(* Logix 5000 project; controller reto3 vendor 1 type 14 code 156 rev 30.11; software revision 30.00 *)

TASK MainTask (continuous, watchdog 500 ms) : MainProgram

MODULES
   Local : vendor 1 type 14 code 156 (Compact 0, rev 30.11)
      DI_4 : 1769-IQ16 (Compact 4, rev 1.1, Input RPI 20 ms)
      D0_5 : vendor 1 type 7 code 86 (Compact 5, rev 2.1, Output RPI 20 ms)
END_MODULES

ADD_ON_INSTRUCTION ACT_DE   (* revision 1.0 *)
VAR_INPUT
   PRENDER_DE : BOOL; {required}
END_VAR
VAR_IN_OUT
   CIERRE_DE : BOOL; {required}
   APERTURA_DE : BOOL; {required}
END_VAR
VAR
   TON_APERTURA_DE : TIMER := (PRE := 200); {access None}
   E_PRENDER : BOOL;
END_VAR

ROUTINE Logic   (* ladder *)
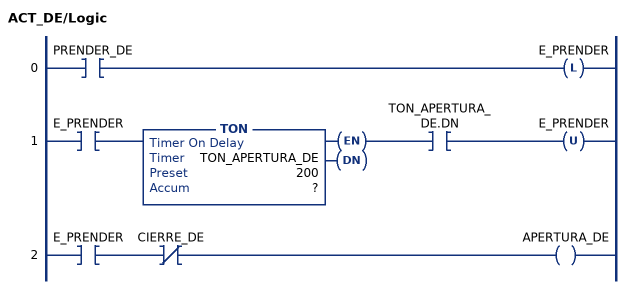
   0: XIC(PRENDER_DE)OTL(E_PRENDER);
   1: XIC(E_PRENDER)TON(TON_APERTURA_DE,?,?)XIC(TON_APERTURA_DE.DN)OTU(E_PRENDER);
   2: XIC(E_PRENDER)XIO(CIERRE_DE)OTE(APERTURA_DE);
END_ROUTINE
END_ADD_ON_INSTRUCTION

ADD_ON_INSTRUCTION CIE_DE   (* revision 1.0 *)
VAR_INPUT
   APAGAR_DE : BOOL; {required}
END_VAR
VAR_IN_OUT
   APERTURA_DE : BOOL; {required}
   CIERRE_DE : BOOL; {required}
END_VAR
VAR
   E_APAGAR : BOOL; {access None}
   TON_CIERRE_dE : TIMER := (PRE := 300); {access None}
END_VAR

ROUTINE Logic   (* ladder *)
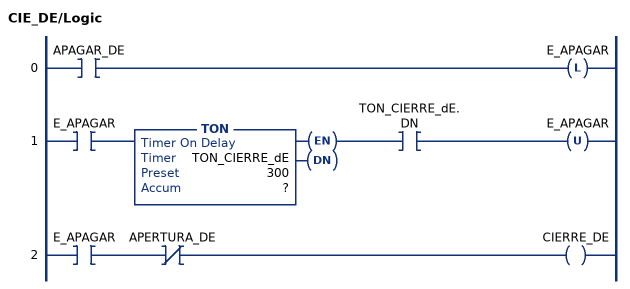
   0: XIC(APAGAR_DE)OTL(E_APAGAR);
   1: XIC(E_APAGAR)TON(TON_CIERRE_dE,?,?)XIC(TON_CIERRE_dE.DN)OTU(E_APAGAR);
   2: XIC(E_APAGAR)XIO(APERTURA_DE)OTE(CIERRE_DE);
END_ROUTINE
END_ADD_ON_INSTRUCTION

ADD_ON_INSTRUCTION COUNTERS   (* revision 1.0 *)
VAR_IN_OUT
   COUNTER_1 : DINT; {required}
END_VAR
VAR_INPUT
   OUT : BOOL; {required}
END_VAR
VAR_IN_OUT
   COUNTER_2 : DINT; {required}
   COUNTER_3 : DINT; {required}
END_VAR
VAR_INPUT
   IN_1 : BOOL; {access None, required}
   IN_2 : BOOL; {access None, required}
   IN_3 : BOOL; {access None, required}
END_VAR
VAR
   CUP_1 : BOOL; {access None}
   CUP_2 : BOOL; {access None}
   CUP_3 : BOOL; {access None}
   OSF_OB1 : BOOL; {access None}
   OSF_SB1 : BOOL; {access None}
   OSF_OB2 : BOOL; {access None}
   OSF_SB2 : BOOL; {access None}
   OSF_OB3 : BOOL; {access None}
   OSF_SB3 : BOOL; {access None}
   OP : BOOL; {access None}
END_VAR

ROUTINE Logic   (* ladder *)
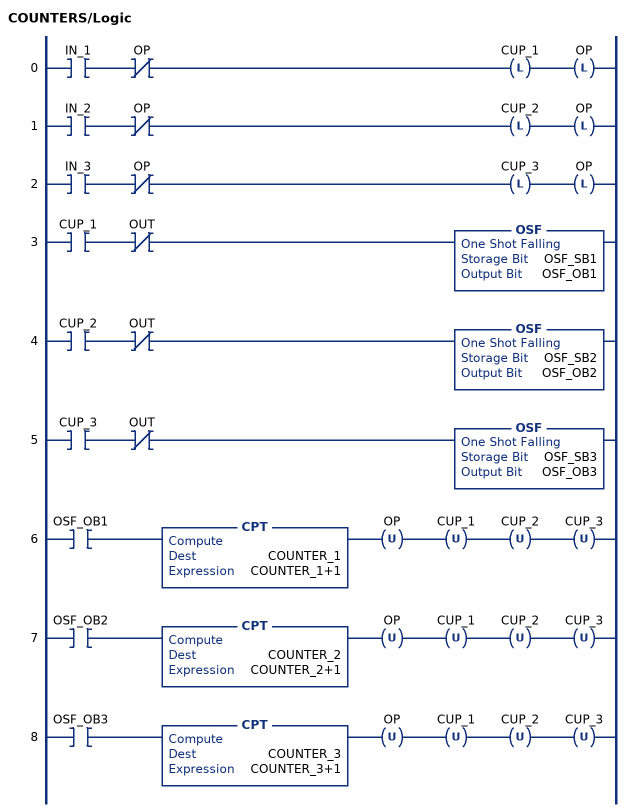
   0: XIC(IN_1)XIO(OP)OTL(CUP_1)OTL(OP);
   1: XIC(IN_2)XIO(OP)OTL(CUP_2)OTL(OP);
   2: XIC(IN_3)XIO(OP)OTL(CUP_3)OTL(OP);
   3: XIC(CUP_1)XIO(OUT)OSF(OSF_SB1,OSF_OB1);
   4: XIC(CUP_2)XIO(OUT)OSF(OSF_SB2,OSF_OB2);
   5: XIC(CUP_3)XIO(OUT)OSF(OSF_SB3,OSF_OB3);
   6: XIC(OSF_OB1)CPT(COUNTER_1,COUNTER_1+1)OTU(OP)OTU(CUP_1)OTU(CUP_2)OTU(CUP_3);
   7: XIC(OSF_OB2)CPT(COUNTER_2,COUNTER_2+1)OTU(OP)OTU(CUP_1)OTU(CUP_2)OTU(CUP_3);
   8: XIC(OSF_OB3)CPT(COUNTER_3,COUNTER_3+1)OTU(OP)OTU(CUP_1)OTU(CUP_2)OTU(CUP_3);
END_ROUTINE
END_ADD_ON_INSTRUCTION

ADD_ON_INSTRUCTION GD_DE   (* revision 1.0 *)
VAR_IN_OUT
   DT : BOOL; {required}
   ABRIR : BOOL; {required}
   CERRAR : BOOL; {required}
END_VAR
VAR
   ONS_DT : BOOL; {access None}
   ON_DE : BOOL; {access None}
   ACT_DE : ACT_DE; {access None}
   CIE_DE : CIE_DE; {access None}
   ONS_DT_NEG : BOOL; {access None}
   OFF_DE : BOOL; {access None}
END_VAR

ROUTINE Logic   (* ladder *)
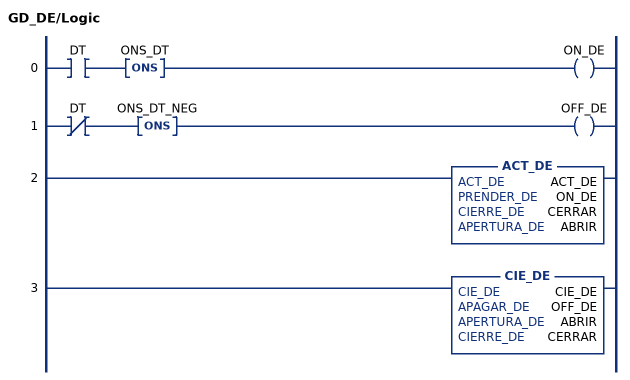
   0: XIC(DT)ONS(ONS_DT)OTE(ON_DE);
   1: XIO(DT)ONS(ONS_DT_NEG)OTE(OFF_DE);
   2: ACT_DE(ACT_DE,ON_DE,CERRAR,ABRIR);
   3: CIE_DE(CIE_DE,OFF_DE,ABRIR,CERRAR);
END_ROUTINE
END_ADD_ON_INSTRUCTION

ADD_ON_INSTRUCTION GD_SE   (* revision 1.0 *)
// Gemelo digital Simple acción/efecto
VAR_IN_OUT
   DT : BOOL; {required}
   RA : BOOL; {required}   // Real Actuator
END_VAR

ROUTINE Logic   (* ladder *)
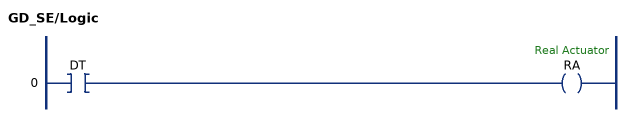
   0: XIC(DT)OTE(RA);
END_ROUTINE
END_ADD_ON_INSTRUCTION

ADD_ON_INSTRUCTION ITEM_DETECTED   (* revision 1.0 *)
VAR_OUTPUT
   DETECTED_1 : BOOL; {access None, required}   // METAL
   DETECTED_2 : BOOL; {access None, required}   // BLUE
   DETECTED_3 : BOOL; {access None, required}   // GREEN
END_VAR
VAR_INPUT
   VISION_SENSOR : DINT; {access None, required}
END_VAR
VAR_IN_OUT
   CONVEYOR : BOOL; {required}
   E0 : BOOL; {required}
END_VAR
VAR
   DETECT : BOOL; {access None}
END_VAR

ROUTINE Logic   (* ladder *)
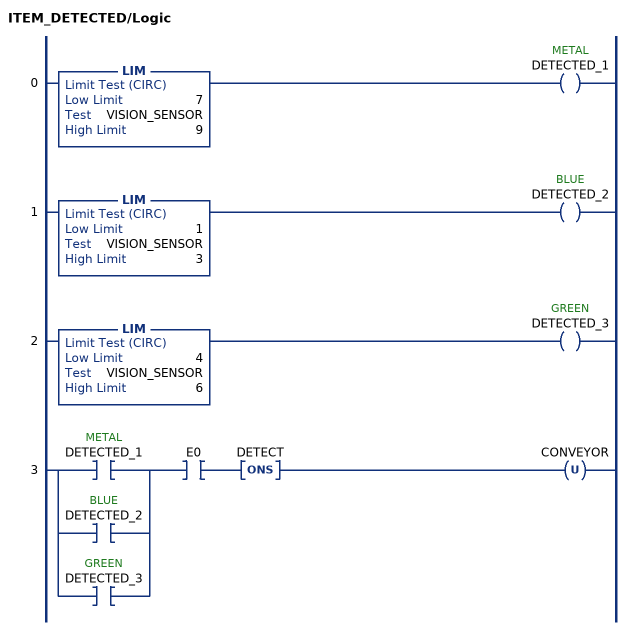
   0: LIM(7,VISION_SENSOR,9)OTE(DETECTED_1);
   1: LIM(1,VISION_SENSOR,3)OTE(DETECTED_2);
   2: LIM(4,VISION_SENSOR,6)OTE(DETECTED_3);
   3: [XIC(DETECTED_1) ,[XIC(DETECTED_2) ,XIC(DETECTED_3) ] ]XIC(E0)ONS(DETECT)OTU(CONVEYOR);
END_ROUTINE
END_ADD_ON_INSTRUCTION

ADD_ON_INSTRUCTION ON_OFF   (* revision 1.0 *)
VAR_INPUT
   ON : BOOL; {required}
   OFF : BOOL; {required}
END_VAR
VAR_IN_OUT
   CONV_1 : BOOL; {required}   // CONVEYOR_1
   CONV_2 : BOOL; {required}   // CONVEYOR_2
   GD_IN_4 : BOOL; {required}
   GD_OUT_0 : BOOL; {required}
   GD_OUT_2 : BOOL; {required}
   GD_OUT_3 : BOOL; {required}
   GD_OUT_4 : BOOL; {required}
   GD_OUT_5 : BOOL; {required}
   GD_OUT_6 : BOOL; {required}
   GD_OUT_7 : BOOL; {required}
   GD_OUT_11 : BOOL; {required}   // STOP LIGHT
   GD_OUT_9 : BOOL; {required}   // START LIGHT
   GD_IN_2 : BOOL; {required}
   GD_OUT_10 : BOOL; {required}   // RESET LIGHT
   E_ON : BOOL; {required}   // Estado ON
   ON_IOT : BOOL; {required}
   OFF_IOT : BOOL; {required}
   GD_INT_OUT_0 : DINT; {required}
   GD_INT_OUT_1 : DINT; {required}
   GD_INT_OUT_2 : DINT; {required}
   GD_OUT_8 : BOOL; {required}
   E2 : BOOL; {required}
   E0 : BOOL; {required}
   GD_IN_5 : BOOL; {required}
   RESET_IOT : BOOL; {required}
   INIT_3 : BOOL; {required}
   INIT_2 : BOOL; {required}
   INIT_1 : BOOL; {required}
END_VAR
VAR
   ONS_ON : BOOL; {access None}
   E_OFF : BOOL; {access None}   // Estado OFF
   ONS_OFF : BOOL; {access None}
   RESET : RESET_ACTS; {access None}
   ON_S : BOOL; {access None}
   OFF_S : BOOL; {access None}
   RES_CONTS : RESET_COUNTERS; {access None}
   ONS_ON_IOT : BOOL; {access None}
   ONS_OFF_IOT : BOOL; {access None}
END_VAR

ROUTINE Logic   (* ladder *)
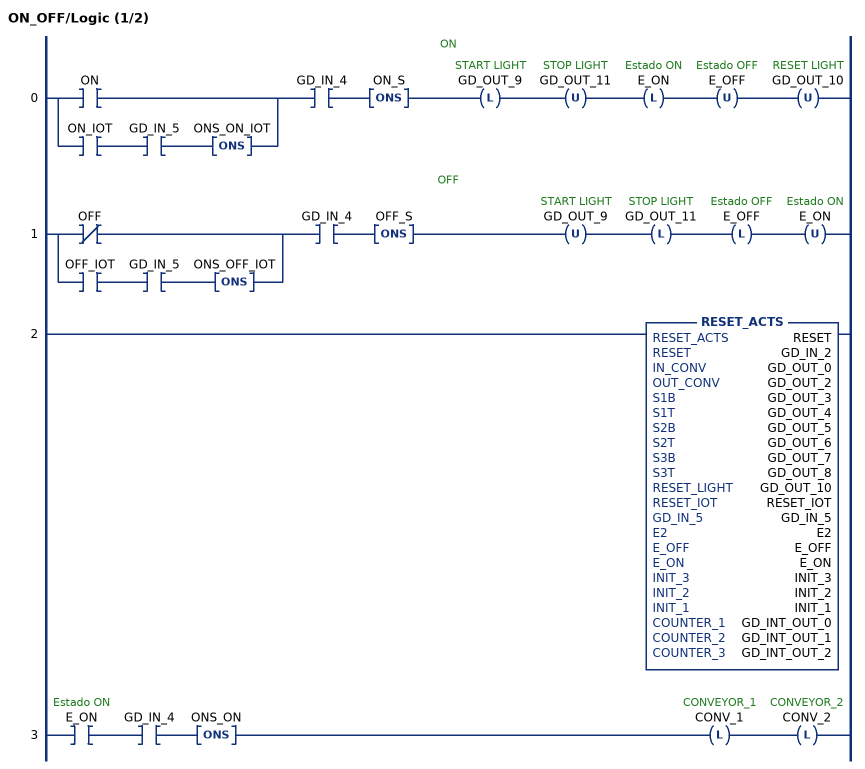
   // ON
   0: [XIC(ON) ,XIC(ON_IOT) XIC(GD_IN_5) ONS(ONS_ON_IOT) ]XIC(GD_IN_4)ONS(ON_S)OTL(GD_OUT_9)OTU(GD_OUT_11)OTL(E_ON)OTU(E_OFF)OTU(GD_OUT_10);
   // OFF
   1: [XIO(OFF) ,XIC(OFF_IOT) XIC(GD_IN_5) ONS(ONS_OFF_IOT) ]XIC(GD_IN_4)ONS(OFF_S)OTU(GD_OUT_9)OTL(GD_OUT_11)OTL(E_OFF)OTU(E_ON);
   2: RESET_ACTS(RESET,GD_IN_2,GD_OUT_0,GD_OUT_2,GD_OUT_3,GD_OUT_4,GD_OUT_5,GD_OUT_6,GD_OUT_7,GD_OUT_8,GD_OUT_10,RESET_IOT,GD_IN_5,E2,E_OFF,E_ON,INIT_3,INIT_2,INIT_1,GD_INT_OUT_0,GD_INT_OUT_1,GD_INT_OUT_2);
   3: XIC(E_ON)XIC(GD_IN_4)ONS(ONS_ON)OTL(CONV_1)OTL(CONV_2);
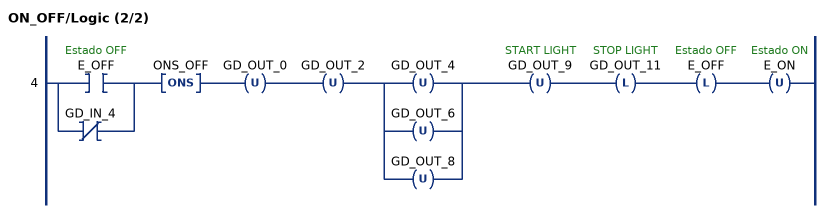
   4: [XIC(E_OFF) ,XIO(GD_IN_4) ]ONS(ONS_OFF)OTU(GD_OUT_0)OTU(GD_OUT_2)[OTU(GD_OUT_4) ,[OTU(GD_OUT_6) ,OTU(GD_OUT_8) ] ]OTU(GD_OUT_9)OTL(GD_OUT_11)OTL(E_OFF)OTU(E_ON);
END_ROUTINE
END_ADD_ON_INSTRUCTION

ADD_ON_INSTRUCTION RESET_ACTS   (* revision 1.0 *)
VAR_IN_OUT
   RESET : BOOL; {required}   // RESET BUTTON
   IN_CONV : BOOL; {required}
   OUT_CONV : BOOL; {required}
   S1B : BOOL; {required}   // Sorter 1 belt
   S1T : BOOL; {required}   // Sorter 1 turn
   S2B : BOOL; {required}
   S2T : BOOL; {required}
   S3B : BOOL; {required}
   S3T : BOOL; {required}
   RESET_LIGHT : BOOL; {required}
   RESET_IOT : BOOL; {required}
   GD_IN_5 : BOOL; {required}   // AUTO
   E2 : BOOL; {required}
   E_OFF : BOOL; {required}
   E_ON : BOOL; {required}
   INIT_3 : BOOL; {required}
   INIT_2 : BOOL; {required}
   INIT_1 : BOOL; {required}
   COUNTER_1 : DINT; {required}
   COUNTER_2 : DINT; {required}
   COUNTER_3 : DINT; {required}
END_VAR
VAR
   ONS_RESET_IOT : BOOL; {access None}
END_VAR

ROUTINE Logic   (* ladder *)
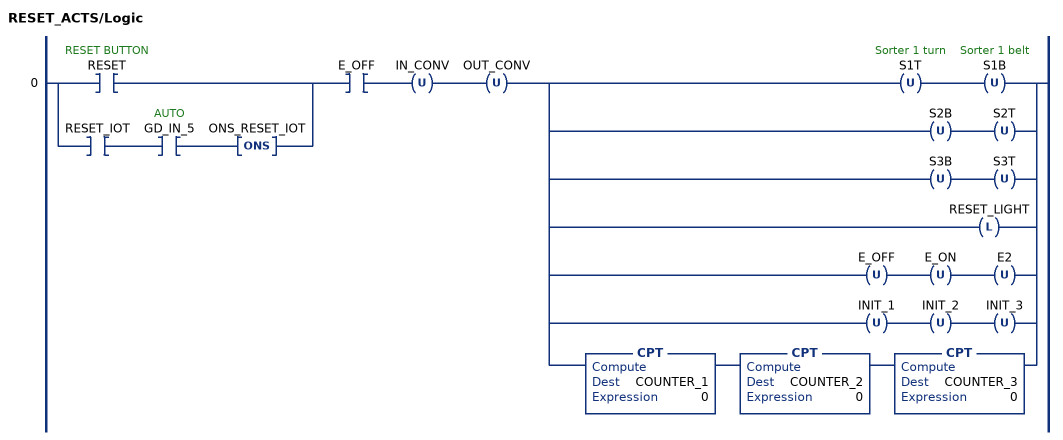
   0: [XIC(RESET) ,XIC(RESET_IOT) XIC(GD_IN_5) ONS(ONS_RESET_IOT) ]XIC(E_OFF)OTU(IN_CONV)OTU(OUT_CONV)[[[OTU(S1T) OTU(S1B) ,[OTU(S2B) OTU(S2T) ,[OTU(S3B) OTU(S3T) ,OTL(RESET_LIGHT) ] ] ] ,[OTU(E_OFF) OTU(E_ON) OTU(E2) ,OTU(INIT_1) OTU(INIT_2) OTU(INIT_3) ] ] ,CPT(COUNTER_1,0) CPT(COUNTER_2,0) CPT(COUNTER_3,0) ];
END_ROUTINE
END_ADD_ON_INSTRUCTION

ADD_ON_INSTRUCTION RESET_COUNTERS   (* revision 1.0 *)
VAR_IN_OUT
   RESET : BOOL; {required}
   COUNTER_1 : DINT; {required}
   COUNTER_2 : DINT; {required}
   COUNTER_3 : DINT; {required}
   RESET_IOT : BOOL; {required}
   GD_IN_5 : BOOL; {required}
   E_OFF : BOOL; {required}
   OFF : BOOL; {required}
END_VAR

ROUTINE Logic   (* ladder *)
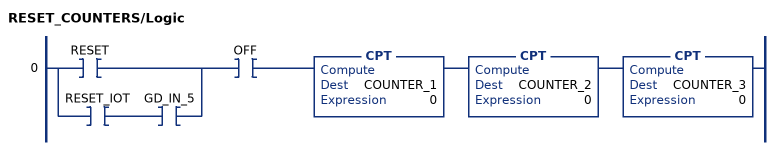
   0: [XIC(RESET) ,XIC(RESET_IOT) XIC(GD_IN_5) ]XIC(OFF)CPT(COUNTER_1,0)CPT(COUNTER_2,0)CPT(COUNTER_3,0);
END_ROUTINE
END_ADD_ON_INSTRUCTION

ADD_ON_INSTRUCTION SORT_X   (* revision 1.0 *)
// MOVE TURN & BELT
VAR_IN_OUT
   TURN : BOOL; {required}   // X TURN
   BELT : BOOL; {required}   // X BELT
END_VAR
VAR_INPUT
   ACTIVATE : BOOL; {access None, required}   // ACTIVATE ROUTINE
   STOP : BOOL; {required}   // STOP TURN & BELT
END_VAR
VAR_IN_OUT
   E2 : BOOL; {required}   // ETAPA SORTING
   ENT_CON : BOOL; {required}   // ENTRY CONVEYOR
   E0 : BOOL; {required}   // ENCENDIDO
END_VAR
VAR
   OSF_STOP : BOOL; {access None}
   OSF_STOP_BIT : BOOL; {access None}
   ONS_SORT : BOOL; {access None}
END_VAR

ROUTINE Logic   (* ladder *)
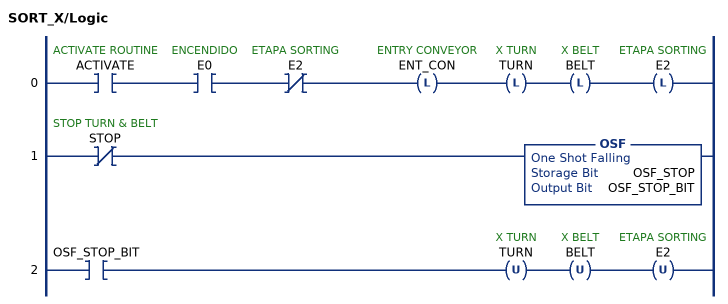
   0: XIC(ACTIVATE)XIC(E0)XIO(E2)OTL(ENT_CON)OTL(TURN)OTL(BELT)OTL(E2);
   1: XIO(STOP)OSF(OSF_STOP,OSF_STOP_BIT);
   2: XIC(OSF_STOP_BIT)OTU(TURN)OTU(BELT)OTU(E2);
END_ROUTINE
END_ADD_ON_INSTRUCTION

VAR_GLOBAL   (* controller tags *)
   CIL_DE_AB : ALIAS FOR Local:5:O.Data.4;
   CIL_DE_CI : ALIAS FOR Local:5:O.Data.5;
   CIL_DE_GD : GD_DE;
   CIL_SE : ALIAS FOR Local:5:O.Data.6;
   CIL_SE_GD : GD_SE;
   COUNTERS : COUNTERS;
   E0 : BOOL;   // Encendido
   E2 : BOOL;   // ETAPA 2
   EMSTOP : RESET_ACTS;
   GD_IN_0 : BOOL;   // At exit
   GD_IN_1 : BOOL;   // START
   GD_IN_2 : BOOL;   // RESET
   GD_IN_3 : BOOL;   // STOP
   GD_IN_4 : BOOL;   // EMERGENCY STOP
   GD_IN_5 : BOOL;   // AUTO
   GD_INT_IN_0 : DINT;   // VISION SENSOR
   GD_INT_OUT_0 : DINT;   // COUNTER 1
   GD_INT_OUT_1 : DINT;   // COUNTER 2
   GD_INT_OUT_2 : DINT;   // COUNTER 3
   GD_OUT_0 : BOOL;   // ENTRY CONVEYOR
   GD_OUT_1 : BOOL;   // STOP BLADE
   GD_OUT_10 : BOOL;   // RESET LIGHT
   GD_OUT_11 : BOOL;   // STOP LIGHT
   GD_OUT_2 : BOOL;   // EXIT CONVEYOR
   GD_OUT_3 : BOOL;   // SORTER 1 TURN
   GD_OUT_4 : BOOL;   // SORTER 1 BELT
   GD_OUT_5 : BOOL;   // SORTER 2 TURN
   GD_OUT_6 : BOOL;   // SORTER 2 BELT
   GD_OUT_7 : BOOL;   // SORTER 3 TURN
   GD_OUT_8 : BOOL;   // SORTER 3 BELT
   GD_OUT_9 : BOOL;   // START LIGHT
   INIT_SORT_1 : BOOL;
   INIT_SORT_2 : BOOL;
   INIT_SORT_3 : BOOL;
   IT_DE_1 : ITEM_DETECTED;
   Motor : ALIAS FOR Local:5:O.Data.0;
   Motor_GD : GD_SE;
   OFF_IOT : BOOL;
   ON_IOT : BOOL;
   ON_OFF : ON_OFF;
   ONS_SORT : BOOL;
   RESET_IOT : BOOL;
   SORT_1 : SORT_X;
   SORT_2 : SORT_X;
   SORT_3 : SORT_X;
   TB_0 : BOOL;
   TB_1 : BOOL;
END_VAR

PROGRAM MainProgram   (* main routine MainRoutine *)

ROUTINE COMMENTS   (* ladder *)
END_ROUTINE

ROUTINE MainRoutine   (* ladder *)
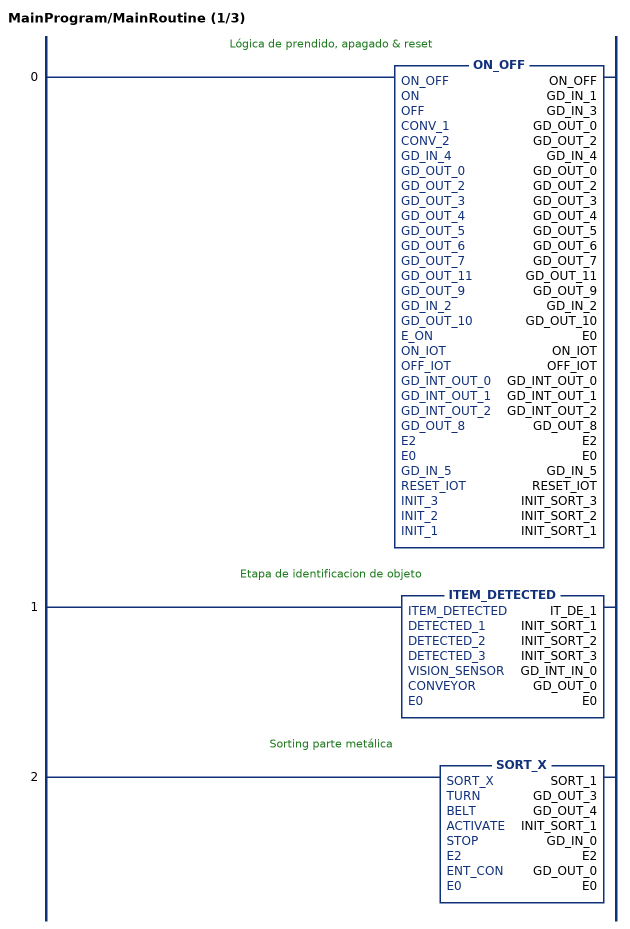
   // Lógica de prendido, apagado & reset
   0: ON_OFF(ON_OFF,GD_IN_1,GD_IN_3,GD_OUT_0,GD_OUT_2,GD_IN_4,GD_OUT_0,GD_OUT_2,GD_OUT_3,GD_OUT_4,GD_OUT_5,GD_OUT_6,GD_OUT_7,GD_OUT_11,GD_OUT_9,GD_IN_2,GD_OUT_10,E0,ON_IOT,OFF_IOT,GD_INT_OUT_0,GD_INT_OUT_1,GD_INT_OUT_2,GD_OUT_8,E2,E0,GD_IN_5,RESET_IOT,INIT_SORT_3,INIT_SORT_2,INIT_SORT_1);
   // Etapa de identificacion de objeto
   1: ITEM_DETECTED(IT_DE_1,INIT_SORT_1,INIT_SORT_2,INIT_SORT_3,GD_INT_IN_0,GD_OUT_0,E0);
   // Sorting parte metálica
   2: SORT_X(SORT_1,GD_OUT_3,GD_OUT_4,INIT_SORT_1,GD_IN_0,E2,GD_OUT_0,E0);
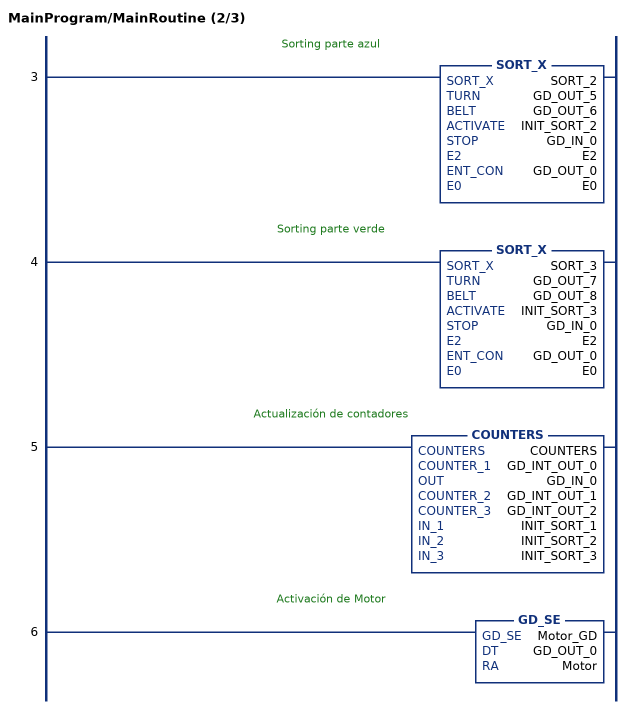
   // Sorting parte azul
   3: SORT_X(SORT_2,GD_OUT_5,GD_OUT_6,INIT_SORT_2,GD_IN_0,E2,GD_OUT_0,E0);
   // Sorting parte verde
   4: SORT_X(SORT_3,GD_OUT_7,GD_OUT_8,INIT_SORT_3,GD_IN_0,E2,GD_OUT_0,E0);
   // Actualización de contadores
   5: COUNTERS(COUNTERS,GD_INT_OUT_0,GD_IN_0,GD_INT_OUT_1,GD_INT_OUT_2,INIT_SORT_1,INIT_SORT_2,INIT_SORT_3);
   // Activación de Motor
   6: GD_SE(Motor_GD,GD_OUT_0,Motor);
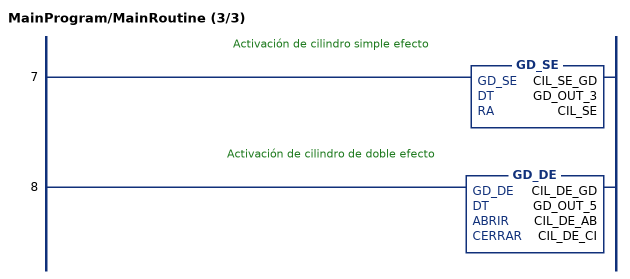
   // Activación de cilindro simple efecto
   7: GD_SE(CIL_SE_GD,GD_OUT_3,CIL_SE);
   // Activación de cilindro de doble efecto
   8: GD_DE(CIL_DE_GD,GD_OUT_5,CIL_DE_AB,CIL_DE_CI);
END_ROUTINE
END_PROGRAM
